(* IEC 61131-3 sources: lc3-ha-sample/src, 6 files *)

(* ---- constants.iecst ---- *)
TYPE
	I2C_ADDRESSES : INT(I2HAE_1 := 16#08, I2HAA_1 := 16#58, PCF8574_OUTPUT_1 := 16#20, PCF8574_INPUT_1 := 16#38);

	MQTT_RC : DINT (OK := 0);
	MQTT_STATE : SINT (INVALID := -1, CONNECTING := 5, CONNECTED := 6);
	MQTT_VALUE : BYTE (DUMMY := 16#31 /* ASCII 1 */);
	MQTT_BROKER : STRING[255] (LOCALHOST := '127.0.0.1');
	MQTT_CLIENTID : STRING[255] (OG_READ := 'OG Read', OG_WRITE := 'OG Write');
	MQTT_TOPICS : STRING[255] (BATH := 'bath', KITCHEN := 'kitchen');
END_TYPE

(* ---- Logic.iecfbd ---- *)
FUNCTION_BLOCK Logic
  {
    height := 50;
    width := 300;
  }

  VAR
    R_TRIG1 : R_TRIG;
    R_TRIG2 : R_TRIG;
  END_VAR
  VAR_INPUT
    signal_bath : BOOL;
    signal_kitchen : BOOL;
    fill_level : UINT;
    analog_input_2 : UINT;
    analog_input_3 : UINT;
    analog_input_4 : UINT;
    analog_input_5 : UINT;
  END_VAR
  VAR_OUTPUT
    light_bath : BOOL;
    light_kitchen : BOOL;
    valve_value : UINT;
    analog_output_2 : UINT;
    analog_output_3 : UINT;
    analog_output_4 : UINT;
    analog_output_5 : UINT;
    light_alarm : BOOL;
  END_VAR

  (*

    // Network 1:
    R_TRIG1(CLK := signal_bath);
    NOT(IN := light_bath, NOT => @C(10).NOT);
    SEL(G := R_TRIG1.Q, IN0 := light_bath, IN1 := @C(10).NOT, SEL => light_bath);

    // Network 2:
    R_TRIG2(CLK := signal_kitchen);
    NOT(IN := light_kitchen, NOT => @C(23).NOT);
    SEL(G := R_TRIG2.Q, IN0 := light_kitchen, IN1 := @C(23).NOT, SEL => light_kitchen);

    // Network 3:
    valve_value := fill_level;
    analog_output_2 := analog_input_2;
    GT(IN1 := fill_level, IN2 := 400, GT => @C(43).GT);
    GT(IN1 := analog_input_2, IN2 := 800, GT => @C(46).GT);
    LT(IN1 := analog_input_2, IN2 := 200, LT => @C(51).LT);
    OR(IN1 := @C(46).GT, IN2 := @C(51).LT, OR => @C(56).OR);
    OR(IN1 := @C(43).GT, IN2 := @C(56).OR, OR => light_alarm);

    // Network 4:
    analog_output_3 := analog_input_3;

    // Network 5:
    analog_output_4 := analog_input_4;

    // Network 6:
    analog_output_5 := analog_input_5;

  *)

  @VF(1) : @E(signal_bath), @R(145.0, 167.0, 140.0, 19.0);
  @VF(2) : @E(light_bath), @R(892.0, 171.0, 140.0, 19.0);
  @C(3) : @FB(R_TRIG1), @R(430.0, 170.0, 140.0, 18.5), @I(@N(CLK), @L(9.5)), @O(@N(Q), @R(9.5));
  @C(5) : @F(SEL), @R(660.0, 170.0, 120.0, 58.0), BOOL, @I(@N(G), @L(9.5)), @I(@N(IN0), @L(29.5)), @I(@N(IN1), @L(49.5)), @O(@N(SEL), @R(9.5));
  @VF(8) : @E(light_bath), @R(430.0, 190.0, 140.0, 19.0);
  @VF(12) : @E(light_bath), @R(430.0, 210.0, 140.0, 19.0);
  @C(10) : @F(NOT), @R(580.0, 213.0, 60.0, 18.5), BOOL, @I(@N(IN), @L(9.5)), @O(@N(NOT), @R(9.5));
  @VF(14) : @E(light_kitchen), @R(903.8, 314.9, 140.0, 19.0);
  @VF(15) : @E(signal_kitchen), @R(140.0, 310.0, 140.0, 19.0);
  @C(16) : @FB(R_TRIG2), @R(430.0, 310.0, 140.0, 18.5), @I(@N(CLK), @L(9.5)), @O(@N(Q), @R(9.5));
  @C(18) : @F(SEL), @R(660.0, 310.0, 120.0, 58.0), BOOL, @I(@N(G), @L(9.5)), @I(@N(IN0), @L(29.5)), @I(@N(IN1), @L(49.5)), @O(@N(SEL), @R(9.5));
  @VF(21) : @E(light_kitchen), @R(427.6, 331.1, 140.0, 19.0);
  @VF(22) : @E(light_kitchen), @R(430.0, 360.0, 140.0, 19.0);
  @C(23) : @F(NOT), @R(580.0, 360.0, 60.0, 18.5), BOOL, @I(@N(IN), @L(9.5)), @O(@N(NOT), @R(9.5));
  @VF(27) : @E(fill_level), @R(150.0, 490.0, 140.0, 19.0);
  @VF(28) : @E(valve_value), @R(900.0, 580.0, 140.0, 19.0);
  @VF(30) : @E(analog_input_2), @R(147.0, 636.4, 140.0, 19.0);
  @VF(31) : @E(analog_input_3), @R(150.0, 840.0, 140.0, 19.0);
  @VF(32) : @E(analog_input_4), @R(150.0, 860.0, 140.0, 19.0);
  @VF(33) : @E(analog_input_5), @R(150.0, 880.0, 140.0, 19.0);
  @VF(34) : @E(analog_output_2), @R(900.0, 690.0, 140.0, 19.0);
  @VF(35) : @E(analog_output_3), @R(900.0, 840.0, 140.0, 19.0);
  @VF(36) : @E(analog_output_4), @R(900.0, 860.0, 140.0, 19.0);
  @VF(37) : @E(analog_output_5), @R(900.0, 880.0, 140.0, 19.0);
  @VF(42) : @E(light_alarm), @R(900.0, 490.0, 140.0, 19.0);
  @C(43) : @F(GT), @R(690.0, 490.0, 40.0, 38.0), UINT, @I(@N(IN1), @L(9.5)), @I(@N(IN2), @L(29.5)), @O(@N(GT), @R(9.5));
  @VF(44) : @E(400), @R(150.0, 510.0, 140.0, 19.0), UINT;
  @C(46) : @F(GT), @R(401.0, 632.1, 40.0, 38.0), UINT, @I(@N(IN1), @L(9.5)), @I(@N(IN2), @L(29.5)), @O(@N(GT), @R(9.5));
  @VF(47) : @E(800), @R(148.0, 655.4, 140.0, 19.0), UINT;
  @C(49) : @F(OR), @R(820.0, 490.0, 40.0, 38.0), BOOL, @I(@N(IN1), @L(9.5)), @I(@N(IN2), @L(29.5)), @O(@N(OR), @R(9.5));
  @C(51) : @F(LT), @R(400.0, 730.0, 40.0, 38.0), UINT, @I(@N(IN1), @L(9.5)), @I(@N(IN2), @L(29.5)), @O(@N(LT), @R(9.5));
  @VF(54) : @E(200), @R(150.0, 750.0, 140.0, 19.0), UINT;
  @C(56) : @F(OR), @R(540.0, 630.0, 40.0, 38.0), BOOL, @I(@N(IN1), @L(9.5)), @I(@N(IN2), @L(29.5)), @O(@N(OR), @R(9.5));
  @CP(53) : 331.0, 645.9;
  @CP(60) : 331.0, 696.5;
  @CP(61) : 329.0, 499.5;

  @G(4) :
     @L(@VF(1).o, @C(3).CLK)
    ;
  @G(6) :
     @L(@C(3).Q, @C(5).G)
    ;
  @G(7) :
     @L(@C(5).SEL, @VF(2).i)
    ;
  @G(9) :
     @L(@VF(8).o, @C(5).IN0)
    ;
  @G(11) :
     @L(@VF(12).o, @C(10).IN)
    ;
  @G(13) :
     @L(@C(10).NOT, @C(5).IN1)
    ;
  @G(17) :
     @L(@VF(15).o, @C(16).CLK)
    ;
  @G(19) :
     @L(@C(16).Q, @C(18).G)
    ;
  @G(20) :
     @L(@C(18).SEL, @VF(14).i)
    ;
  @G(24) :
     @L(@VF(22).o, @C(23).IN)
    ;
  @G(25) :
     @L(@C(23).NOT, @C(18).IN1)
    ;
  @G(26) :
     @L(@VF(21).o, @C(18).IN0)
    ;
  @G(39) :
     @L(@VF(31).o, @VF(35).i)
    ;
  @G(40) :
     @L(@VF(32).o, @VF(36).i)
    ;
  @G(41) :
     @L(@VF(33).o, @VF(37).i)
    ;
  @G(29) :
     @L(@VF(27).o, @CP(61)),
     @L(@CP(61), @C(43).IN1),
     @L(@CP(61), @VF(28).i)
    ;
  @G(45) :
     @L(@VF(44).o, @C(43).IN2)
    ;
  @G(38) :
     @L(@VF(30).o, @CP(53)),
     @L(@CP(53), @C(46).IN1),
     @L(@CP(53), @CP(60)),
     @L(@CP(60), @C(51).IN1),
     @L(@CP(60), @VF(34).i)
    ;
  @G(48) :
     @L(@VF(47).o, @C(46).IN2)
    ;
  @G(50) :
     @L(@C(43).GT, @C(49).IN1)
    ;
  @G(52) :
     @L(@C(49).OR, @VF(42).i)
    ;
  @G(55) :
     @L(@VF(54).o, @C(51).IN2)
    ;
  @G(57) :
     @L(@C(46).GT, @C(56).IN1)
    ;
  @G(58) :
     @L(@C(51).LT, @C(56).IN2)
    ;
  @G(59) :
     @L(@C(56).OR, @C(49).IN2)
    ;
END_FUNCTION_BLOCK

(* ---- readinputs.iecst ---- *)
FUNCTION_BLOCK ReadInputs
	{
		height := 250;
		width := 300;
	}
	VAR_OUTPUT
		digital_1_1 : BOOL;
		digital_1_2 : BOOL;
		digital_1_3 : BOOL;
		digital_1_4 : BOOL;
		digital_1_5 : BOOL;
		digital_1_6 : BOOL;
		digital_1_7 : BOOL;
		digital_1_8 : BOOL;

		analog_1_1 : UINT;
		analog_1_2 : UINT;
		analog_1_3 : UINT;
		analog_1_4 : UINT;
		analog_1_5 : UINT;

		mqtt_1_1 : BOOL;
		mqtt_1_2 : BOOL;
		mqtt_1_3 : BOOL;
		mqtt_1_4 : BOOL;
	END_VAR

	VAR
		i2c_handle : DINT := -1;
		pin_values_1 : ARRAY [0..7] OF BOOL;

		mqtt_state : MQTT_STATE := MQTT_STATE#INVALID;
		mqtt_rc : DINT;
		mqtt_handle : DINT := -1;
		mqtt_subscribed : BOOL;
		mqtt_payload : ARRAY [0..0] OF BYTE;
		mqtt_payload_len_received : DINT;
	END_VAR

	/* I2C */
	IF i2c_handle < 0 THEN
		i2c_handle := I2C_open(bus_id := 1);
	ELSE
		pin_values_1 := I2C_PCF8574_read(fd := i2c_handle, address := I2C_ADDRESSES#PCF8574_INPUT_1);
		digital_1_1 := pin_values_1[0];
		digital_1_2 := pin_values_1[1];
		digital_1_3 := pin_values_1[2];
		digital_1_4 := pin_values_1[3];
		digital_1_5 := pin_values_1[4];
		digital_1_6 := pin_values_1[5];
		digital_1_7 := pin_values_1[6];
		digital_1_8 := pin_values_1[7];

		I2C_I2HAE_read(fd := i2c_handle, address := I2C_ADDRESSES#I2HAE_1,
			values[0] => analog_1_1,
			values[1] => analog_1_2,
			values[2] => analog_1_3,
			values[3] => analog_1_4,
			values[4] => analog_1_5
		);
	END_IF;

	/* MQTT */
	mqtt_state := MQTT_GetState(ch := mqtt_handle);
	IF mqtt_state <> MQTT_STATE#CONNECTING AND mqtt_state <> MQTT_STATE#CONNECTED THEN
		mqtt_handle := MQTT_Connect(address := MQTT_BROKER#LOCALHOST, clientId := MQTT_CLIENTID#OG_READ);
	END_IF;

	IF mqtt_state = MQTT_STATE#CONNECTED THEN
		IF NOT mqtt_subscribed THEN
			MQTT_Subscribe(ch := mqtt_handle, topic := MQTT_TOPICS#BATH, rc => mqtt_rc);
			mqtt_subscribed := mqtt_rc = MQTT_RC#OK;
		END_IF;
		IF mqtt_subscribed THEN
			MQTT_Receive(ch := mqtt_handle, payload := REF(mqtt_payload[0]), payload_len := TO_DINT(SIZEOF(mqtt_payload)), len => mqtt_payload_len_received, rc => mqtt_rc);
			mqtt_1_1 := mqtt_rc = MQTT_RC#OK AND mqtt_payload[0] = MQTT_VALUE#DUMMY;
		END_IF;
	ELSE
		mqtt_subscribed := FALSE;
	END_IF;
END_FUNCTION_BLOCK

(* ---- writeoutputs.iecst ---- *)
FUNCTION_BLOCK WriteOutputs
  {
    height := 250;
    width := 250;
  }
	VAR_INPUT
		relay_1_1 : BOOL;
		relay_1_2 : BOOL;
		relay_1_3 : BOOL;
		relay_1_4 : BOOL;
		relay_1_5 : BOOL;
		relay_1_6 : BOOL;
		relay_1_7 : BOOL;
		relay_1_8 : BOOL;

		analog_1_1 : UINT;
		analog_1_2 : UINT;
		analog_1_3 : UINT;
		analog_1_4 : UINT;
		analog_1_5 : UINT;

		mqtt_1_1 : BOOL;
		mqtt_1_2 : BOOL;
		mqtt_1_3 : BOOL;
		mqtt_1_4 : BOOL;
	END_VAR

	VAR
		i2c_handle : DINT := -1;
		pin_values_1 : ARRAY[0..7] OF BOOL;
		analog_values_1 : ARRAY[0..4] OF UINT;
		mqtt_state : MQTT_STATE := MQTT_STATE#INVALID;
		mqtt_rc : DINT := -1;
		mqtt_handle : DINT := -1;
		mqtt_payload : ARRAY [0..0] OF BYTE := [ MQTT_VALUE#DUMMY ];
	END_VAR

	/* I2C */
	IF i2c_handle < 0 THEN
		i2c_handle := I2C_open(bus_id := 1);
	ELSE
		pin_values_1[0] := relay_1_1;
		pin_values_1[1] := relay_1_2;
		pin_values_1[2] := relay_1_3;
		pin_values_1[3] := relay_1_4;
		pin_values_1[4] := relay_1_5;
		pin_values_1[5] := relay_1_6;
		pin_values_1[6] := relay_1_7;
		pin_values_1[7] := relay_1_8;
		I2C_PCF8574_write(fd := i2c_handle, address := I2C_ADDRESSES#PCF8574_OUTPUT_1, pin_values := pin_values_1);

		analog_values_1[0] := analog_1_1;
		analog_values_1[1] := analog_1_2;
		analog_values_1[2] := analog_1_3;
		analog_values_1[3] := analog_1_4;
		analog_values_1[4] := analog_1_5;
		I2C_I2HAA_write(fd := i2c_handle, address := I2C_ADDRESSES#I2HAA_1, values := analog_values_1);
	END_IF;

	/* MQTT */
	mqtt_state := MQTT_GetState(ch := mqtt_handle, rc => mqtt_rc, ENO => ENO);
	IF mqtt_state <> MQTT_STATE#CONNECTING AND mqtt_state <> MQTT_STATE#CONNECTED THEN
		mqtt_handle := MQTT_CONNECT(address := MQTT_BROKER#LOCALHOST, clientId := MQTT_CLIENTID#OG_WRITE, ENO => ENO);
	END_IF;
	IF ENO and mqtt_state = MQTT_STATE#CONNECTED THEN
		IF mqtt_1_1 THEN
			MQTT_Publish(ch := mqtt_handle, topic := MQTT_TOPICS#KITCHEN, payload := REF(mqtt_payload[0]), len := TO_DINT(SIZEOF(mqtt_payload)), rc => mqtt_rc);
		END_IF;
	END_IF;
END_FUNCTION_BLOCK

(* ---- HomeAutomationHardware.iecfbd ---- *)
PROGRAM HomeAutomationHardware
  VAR
    ReadInputs1 : ReadInputs;
    WriteOutputs1 : WriteOutputs;
    Logic1 : Logic;
    R_TRIG1 : R_TRIG;
    F_TRIG1 : F_TRIG;
  END_VAR

  (*

    // Network 1:
    ReadInputs1();
    OR(IN1 := ReadInputs1.digital_1_1, IN2 := ReadInputs1.mqtt_1_1, OR => @C(4).OR);
    Logic1(signal_bath := @C(4).OR, signal_kitchen := ReadInputs1.digital_1_2, fill_level := ReadInputs1.analog_1_1, analog_input_2 := ReadInputs1.analog_1_2, analog_input_3 := ReadInputs1.analog_1_3, analog_input_4 := ReadInputs1.analog_1_4, analog_input_5 := ReadInputs1.analog_1_5);
    R_TRIG1(CLK := Logic1.light_kitchen);
    F_TRIG1(CLK := Logic1.light_kitchen);
    OR(IN1 := R_TRIG1.Q, IN2 := F_TRIG1.Q, OR => @C(11).OR);
    WriteOutputs1(relay_1_1 := Logic1.light_bath, relay_1_2 := Logic1.light_alarm, analog_1_1 := Logic1.valve_value, analog_1_2 := Logic1.analog_output_2, analog_1_3 := Logic1.analog_output_3, analog_1_4 := Logic1.analog_output_4, analog_1_5 := Logic1.analog_output_5, mqtt_1_1 := @C(11).OR);

  *)

  @C(4) : @F(OR), @R(577.6, 127.0, 40.0, 38.0), BOOL, @I(@N(IN1), @L(9.5)), @I(@N(IN2), @L(29.5)), @O(@N(OR), @R(9.5));
  @C(9) : @FB(R_TRIG1), @R(1198.9, 383.4, 140.0, 18.5), @I(@N(CLK), @L(9.5)), @O(@N(Q), @R(9.5));
  @C(10) : @FB(F_TRIG1), @R(1200.5, 403.6, 140.0, 18.5), @I(@N(CLK), @L(9.5)), @O(@N(Q), @R(9.5));
  @C(11) : @F(OR), @R(1366.3, 391.1, 40.0, 38.0), BOOL, @I(@N(IN1), @L(9.5)), @I(@N(IN2), @L(29.5)), @O(@N(OR), @R(9.5));
  @C(5) : @FB(ReadInputs1), @R(135.1, 120.4, 300.0, 338.0), @O(@N(digital_1_1), @R(9.5)), @O(@N(digital_1_2), @R(29.5)), @O(@N(digital_1_3), @R(49.5)), @O(@N(digital_1_4), @R(69.5)), @O(@N(digital_1_5), @R(89.5)), @O(@N(digital_1_6), @R(109.5)), @O(@N(digital_1_7), @R(129.5)), @O(@N(digital_1_8), @R(149.5)), @O(@N(analog_1_1), @R(169.5)), @O(@N(analog_1_2), @R(189.5)), @O(@N(analog_1_3), @R(209.5)), @O(@N(analog_1_4), @R(229.5)), @O(@N(analog_1_5), @R(249.5)), @O(@N(mqtt_1_1), @R(269.5)), @O(@N(mqtt_1_2), @R(289.5)), @O(@N(mqtt_1_3), @R(309.5)), @O(@N(mqtt_1_4), @R(329.5));
  @C(1) : @FB(WriteOutputs1), @R(1581.3, 135.0, 250.0, 338.0), @I(@N(relay_1_1), @L(9.5)), @I(@N(relay_1_2), @L(29.5)), @I(@N(relay_1_3), @L(49.5)), @I(@N(relay_1_4), @L(69.5)), @I(@N(relay_1_5), @L(89.5)), @I(@N(relay_1_6), @L(109.5)), @I(@N(relay_1_7), @L(129.5)), @I(@N(relay_1_8), @L(149.5)), @I(@N(analog_1_1), @L(169.5)), @I(@N(analog_1_2), @L(189.5)), @I(@N(analog_1_3), @L(209.5)), @I(@N(analog_1_4), @L(229.5)), @I(@N(analog_1_5), @L(249.5)), @I(@N(mqtt_1_1), @L(269.5)), @I(@N(mqtt_1_2), @L(289.5)), @I(@N(mqtt_1_3), @L(309.5)), @I(@N(mqtt_1_4), @L(329.5));
  @OLT(28) : @R(520.0, 460.0, 80.0, 18.0), @S(@C(5).analog_1_2);
  @OLT(29) : @R(1350.0, 490.0, 80.0, 18.0), @S(@C(10).Q);
  @OLT(31) : @R(1340.0, 320.0, 80.0, 18.0), @S(@C(9).Q);
  @OLT(14) : @R(600.0, 410.0, 80.0, 18.0), @S(@C(5).analog_1_1);
  @C(7) : @FB(Logic1), @R(804.3, 130.2, 300.0, 158.0), @I(@N(signal_bath), @L(9.5)), @I(@N(signal_kitchen), @L(29.5)), @I(@N(fill_level), @L(49.5)), @I(@N(analog_input_2), @L(69.5)), @I(@N(analog_input_3), @L(89.5)), @I(@N(analog_input_4), @L(109.5)), @I(@N(analog_input_5), @L(129.5)), @O(@N(light_bath), @R(9.5)), @O(@N(light_kitchen), @R(29.5)), @O(@N(valve_value), @R(49.5)), @O(@N(analog_output_2), @R(69.5)), @O(@N(analog_output_3), @R(89.5)), @O(@N(analog_output_4), @R(109.5)), @O(@N(analog_output_5), @R(129.5)), @O(@N(light_alarm), @R(149.5));
  @CP(30) : 1151.6, 393.5;

  @G(3) :
     @L(@C(5).digital_1_1, @C(4).IN1)
    ;
  @G(6) :
     @L(@C(5).mqtt_1_1, @C(4).IN2)
    ;
  @G(2) :
     @L(@C(4).OR, @C(7).signal_bath)
    ;
  @G(8) :
     @L(@C(7).light_bath, @C(1).relay_1_1)
    ;
  @G(12) :
     @L(@C(11).OR, @C(1).mqtt_1_1)
    ;
  @G(15) :
     @L(@C(9).Q, @C(11).IN1)
    ;
  @G(16) :
     @L(@C(10).Q, @C(11).IN2)
    ;
  @G(17) :
     @L(@C(5).digital_1_2, @C(7).signal_kitchen)
    ;
  @G(18) :
     @L(@C(5).analog_1_1, @C(7).fill_level)
    ;
  @G(19) :
     @L(@C(7).valve_value, @C(1).analog_1_1)
    ;
  @G(20) :
     @L(@C(5).analog_1_2, @C(7).analog_input_2)
    ;
  @G(21) :
     @L(@C(5).analog_1_3, @C(7).analog_input_3)
    ;
  @G(22) :
     @L(@C(5).analog_1_4, @C(7).analog_input_4)
    ;
  @G(23) :
     @L(@C(5).analog_1_5, @C(7).analog_input_5)
    ;
  @G(24) :
     @L(@C(7).analog_output_2, @C(1).analog_1_2)
    ;
  @G(25) :
     @L(@C(7).analog_output_3, @C(1).analog_1_3)
    ;
  @G(26) :
     @L(@C(7).analog_output_4, @C(1).analog_1_4)
    ;
  @G(27) :
     @L(@C(7).analog_output_5, @C(1).analog_1_5)
    ;
  @G(13) :
     @L(@C(7).light_kitchen, @CP(30)),
     @L(@CP(30), @C(10).CLK),
     @L(@CP(30), @C(9).CLK)
    ;
  @G(32) :
     @L(@C(7).light_alarm, @C(1).relay_1_2)
    ;
END_PROGRAM

(* ---- HomeAutomationSimulation.iecst ---- *)
/**
 * Too simple for being implemented in FBD
 */
PROGRAM HomeAutomationSimulation
	VAR
		logic : Logic;
	END_VAR

	logic();

END_PROGRAM
